Fanuc KAREL source: compact_preamble.KL

PROGRAM KD00017
%NOLOCKGROUP
VAR
I:INTEGER;J:INTEGER;B:BOOLEAN;R:REAL;S : STRING[80]
BEGIN
I=0
CONNECT TIMER TO I
DISCONNECT TIMER I
END KD00017
